///EL2258 | XFC, 8-channel digital output terminal with time stamp
FUNCTION_BLOCK EL2258_v0_00

END_FUNCTION_BLOCK

(* stored: Version 1.1.0.1, ProductVersion 3.1.4022.6
   POU EL2258_v0_00: Id {bc3f9533-dbfa-4783-a124-6afca138fe1c}, SpecialFunc None *)
